VAR_GLOBAL
	L_Licht : BOOL;
	L_EinbruchBild : STRING;
	WetterBild : STRING := BildWolke;
	
	Besucher : INT;
	Alarm : BOOL;
	heizung_SIM : INT;
	
	Sim_Haus_Glocke : BOOL;
	Sim_Haus_Alarm : BOOL;
	Sim_Haus_ResetAlarm: BOOL;
END_VAR

(* stored: Version 1.1.0.1, ProductVersion 3.1.4018.5
   GVL HausSim: Id {374952b0-c91d-4138-9ac9-fe1efef1c703} *)
